Yaskawa INFORM job: OK_R2_O27-28(-60,-90)OKKR.JBI

/JOB
//NAME OK_R2_O27-28(-60,-90)OKKR
///FOLDERNAME X4
//POS
///NPOS 257,257,257,8,0,0
///TOOL 0
///POSTYPE PULSE
///PULSE
C00000=-3986,-112829,-111510,7465,89684,-2966
C00001=-141364,-59194,-77930,23847,91990,-48786
C00002=-141063,-58232,-69990,23735,87869,-49501
C00003=-140498,-58627,-69073,23636,87005,-49471
C00004=-140498,-58696,-68045,23642,86390,-49593
C00005=-140498,-58689,-68203,23640,86482,-49574
C00006=-139283,-59279,-68522,23418,86041,-49222
C00007=-140498,-58679,-68345,23640,86568,-49558
C00008=-140498,-58443,-70820,23629,88081,-49258
C00009=-127873,-62764,-73114,21064,83986,-45532
C00010=-126392,-63087,-72194,20752,82931,-45191
C00011=-125308,-63227,-72265,20505,82639,-44857
C00012=-125876,-63157,-72230,20635,82791,-45032
C00013=-125876,-63224,-70878,20668,81976,-45171
C00014=-126013,-60778,-71127,20647,83335,-44988
C00015=-126013,-60882,-69659,20681,82436,-45141
C00016=-127370,-60434,-72326,20932,84528,-45261
C00017=-126178,-37548,-64770,20629,90906,-43754
C00018=-125360,-36121,-63262,20430,90533,-43541
C00019=-124562,-36215,-63320,20235,90337,-43305
C00020=-125156,-36149,-63276,20379,90482,-43482
C00021=-125105,-34567,-61617,20363,90274,-43498
C00022=-125156,-36149,-63276,20379,90482,-43482
C00023=-135815,-54991,-80141,22838,93753,-46517
C00024=-126128,-100939,-98074,-7833,62391,34723
C00025=-121019,-58487,-70527,-23750,81541,54822
C00026=-122085,-55123,-66318,-23503,80455,54653
C00027=-122085,-55198,-65243,-23545,79813,54780
C00028=-122085,-55189,-65403,-23539,79908,54761
C00029=-123392,-55124,-65366,-23193,79559,54356
C00030=-122085,-54853,-68645,-23426,81902,54365
C00031=-134552,-52582,-66238,-19865,78414,50556
C00032=-135818,-52234,-64976,-19512,77552,50249
C00033=-136587,-51927,-64802,-19268,77420,49997
C00034=-135954,-52181,-64946,-19469,77528,50205
C00035=-135954,-52277,-63949,-19514,76901,50308
C00036=-136080,-52138,-64861,-19432,77470,50170
C00037=-136080,-52251,-63636,-19487,76702,50295
C00038=-135954,-52187,-64889,-19472,77492,50211
C00039=-133506,-28182,-57356,-19912,85326,49780
C00040=-133698,-26913,-56229,-19853,85243,49729
C00041=-134401,-26653,-56048,-19633,85105,49516
C00042=-133766,-26888,-56212,-19832,85229,49708
C00043=-133683,-26061,-55050,-19864,84975,49778
C00044=-133766,-26888,-56212,-19832,85229,49708
C00045=-118022,-32997,-63083,-24386,90185,54129
C00046=-121676,-92941,-80647,-24717,48269,48100
C00047=-126104,-89968,-74727,-22625,45053,46752
C00048=-126437,-97824,-79818,-22747,44125,46828
C00049=-122563,-90224,-74830,-24996,46013,48290
C00050=-126668,-97900,-73203,-24411,40283,47817
C00051=-125704,-63387,-70361,-17497,77836,40931
C00052=-124997,-29881,-53878,-19439,104666,37001
C00053=-125884,-60589,-72245,-19026,100228,37410
C00054=-128512,-118388,-89616,-19043,55419,43468
C00055=-135431,-142346,-71459,-72171,9437,70233
C00056=-131754,-155096,-83372,-71140,11907,70394
C00057=-142652,-70242,-76718,-4199,55092,38367
C00058=-144604,-67983,-72835,-2974,53782,37623
C00059=-145152,-70837,-74169,-2632,53116,37415
C00060=-145458,-72223,-74577,-2444,52646,37302
C00061=-149846,-88596,-70971,7115,30316,34609
C00062=-154437,-99635,-68231,16252,23743,29866
C00063=-154437,-99624,-68210,16257,23736,29864
C00064=-147075,-80257,-74853,-4272,57747,36179
C00065=-135105,-30448,-54067,-19922,99128,39315
C00066=-136639,-45484,-63511,-20526,99341,42271
C00067=-135372,-63496,-79310,-18587,95300,36150
C00068=-132445,-62328,-82142,-19075,98166,36710
C00069=-146017,-78257,-86482,14597,77172,-40405
C00070=-148450,-84312,-78135,27735,61043,-43185
C00071=-146415,-83246,-79022,27034,61486,-42173
C00072=-149676,-80485,-74368,28759,61288,-43622
C00073=-146415,-82526,-75268,27520,59752,-42632
C00074=-148666,-91519,-74847,29905,56218,-44658
C00075=-148661,-91510,-74815,29908,56203,-44660
C00076=-141622,-55635,-68822,15914,88047,-36263
C00077=-139223,-29516,-55234,13545,105159,-43741
C00078=-138881,-22432,-50139,13428,110509,-48714
C00079=-142652,-51115,-68560,12963,107777,-50366
C00080=-150767,-106394,-89377,20632,70658,-55438
C00081=-159311,-126903,-88538,34684,53320,-63895
C00082=-162771,-130732,-86957,36938,52328,-66028
C00083=-169268,-142526,-99377,37807,56354,-67589
C00084=-135427,-86810,-88528,19455,64054,-50570
C00085=-130773,-34503,-67642,16020,92669,-44609
C00086=-128794,-31809,-63686,15472,92294,-44000
C00087=-128893,-32813,-64547,15497,92321,-44030
C00088=-130866,-69048,-76557,19964,64993,-48316
C00089=-131163,-70480,-77226,20153,64757,-48473
C00090=-131351,-74311,-77618,20524,63181,-48835
C00091=-132679,-88532,-78088,22594,56973,-50647
C00092=-132679,-88527,-78070,22596,56965,-50649
C00093=-130794,-63914,-72852,16389,80850,-46075
C00094=-128797,-28836,-55060,14325,107943,-42385
C00095=-129807,-49025,-67626,14097,105546,-43031
C00096=-134716,-44704,-73522,14618,112039,-43955
C00097=-29759,-44704,-73522,14618,112039,-43955
C00098=-57909,-76089,-130518,-12878,65640,73000
C00099=-127209,-68927,-129586,-14791,77681,41071
C00100=-94927,-66213,-124589,-13119,107191,-29169
C00101=-113727,-82793,-127993,9786,99340,-30667
C00102=-113727,-86481,-127524,9719,97186,-30836
C00103=-113727,-85675,-127642,9732,97666,-30798
C00104=-112224,-85220,-127466,9230,97646,-30371
C00105=-92228,-67360,-123883,-12571,107517,-29060
C00106=-93915,-95192,-134825,-11586,99912,-28771
C00107=-93907,-97921,-132985,-11491,97428,-28535
C00108=-94423,-93096,-131262,-11383,98761,-28810
C00109=-93907,-97921,-132985,-11491,97428,-28535
C00110=-98178,-92441,-135596,-10352,101296,-30120
C00111=-110030,-49454,-111281,11211,101949,-41769
C00112=-110030,-52113,-110961,11140,100416,-41912
C00113=-110030,-50840,-111124,11173,101156,-41843
C00114=-108714,-50397,-110891,10661,101109,-41508
C00115=-110030,-50840,-111124,11173,101156,-41843
C00116=-94659,-80928,-124596,-7278,89440,-41621
C00117=-94884,-83616,-122998,-7181,87076,-41547
C00118=-95311,-80232,-121621,-6996,87929,-41716
C00119=-94926,-83537,-124629,-7161,88110,-41617
C00120=-94884,-64304,-125016,-7294,98157,-42187
C00121=-68339,-68740,-122629,-37645,97901,-27341
C00122=-68339,-68740,-122629,-37645,97901,-27341
C00123=-67428,-88828,-131318,-26507,103272,13068
C00124=-71370,-89365,-129778,-25198,101161,12301
C00125=-78547,-84496,-129463,-18628,102671,11282
C00126=-78547,-86342,-129276,-18525,101662,11444
C00127=-78560,-85520,-129334,-18575,102093,11369
C00128=-79372,-81461,-127756,-18419,103003,10989
C00129=-78560,-82342,-129603,-18733,103801,11099
C00130=-72065,-90999,-130386,-24944,100563,12212
C00131=-83791,-78457,-128497,-14695,105981,10194
C00132=-83791,-80329,-128373,-14610,104970,10319
C00133=-83791,-79121,-128456,-14665,105627,10237
C00134=-84464,-75325,-126915,-14548,106502,9937
C00135=-83407,-79441,-129435,-14816,106104,10287
C00136=-72065,-90999,-130386,-24944,100563,12212
C00137=-83702,-92322,-133428,-14376,100027,10952
C00138=-83702,-94820,-133208,-14304,98651,11113
C00139=-83702,-93492,-133334,-14341,99387,11027
C00140=-84690,-87135,-131003,-14116,101025,10548
C00141=-83702,-92262,-133433,-14377,100059,10948
C00142=-70978,-78992,-130158,-26016,106298,11265
C00143=-70978,-75133,-130239,-32870,108132,50816
C00144=-78131,-73748,-122265,-29687,102174,50283
C00145=-78131,-74118,-122214,-29659,101980,50334
C00146=-78131,-76651,-121813,-29472,100626,50691
C00147=-78131,-74997,-122085,-29593,101516,50457
C00148=-79801,-77736,-123237,-28954,100436,50209
C00149=-73940,-85384,-126808,-30662,100615,52053
C00150=-80113,-114247,-134388,-23740,88254,34284
C00151=-81075,-108298,-132442,-23441,89717,33674
C00152=-80541,-110046,-134005,-23615,89911,33813
C00153=-80541,-103654,-135317,-23722,93674,33065
C00154=-68201,-105154,-135623,-27548,96450,36475
C00155=-62711,-72176,-121164,-35654,111043,40715
C00156=-62711,-74449,-120804,-35309,109900,41112
C00157=-62711,-73505,-120963,-35451,110380,40946
C00158=-63747,-76072,-122060,-35030,109506,40878
C00159=-62711,-70908,-121334,-35852,111664,40494
C00160=-49527,-79873,-125116,-38340,114336,44330
C00161=-57136,-119945,-136347,-29907,93340,40844
C00162=-58022,-116776,-135357,-29743,93940,40370
C00163=-57136,-119945,-136347,-29907,93340,40844
C00164=-54754,-67051,-118805,-40417,118327,44687
C00165=-59603,-68009,-118098,-39014,115880,43853
C00166=-69985,-90348,-127433,-28935,99872,36944
C00167=-57627,-107220,-134942,-31595,99953,40891
C00168=-57921,-110194,-135915,-31186,98692,-1554
C00169=-57134,-101414,-130612,-30299,94100,-6411
C00170=-59324,-101870,-130514,-29608,93156,-6916
C00171=-56722,-67413,-112454,-48445,106979,-15822
C00172=-54266,-64565,-109317,-53003,108151,-17088
C00173=-41269,-82198,-112353,-60396,104555,-10877
C00174=-28361,-73162,-108384,-64272,112863,-9833
C00175=-27672,-73415,-108865,-64508,113328,-9806
C00176=-47228,-89020,-130256,-33764,105577,26890
C00177=-61305,-120775,-136286,-22017,83813,21194
C00178=-54809,-66121,-115305,-41444,115205,18852
C00179=-55914,-62658,-119826,-31689,114363,21910
C00180=-59579,-116943,-133527,-40693,98814,56774
C00181=-59579,-111986,-135330,-41226,101614,55657
C00182=-82689,-64404,-114714,-44753,105294,68555
C00183=-85026,-71008,-115277,-43369,102134,69076
C00184=-83828,-73704,-112663,-46568,100432,69183
C00185=-87462,-56287,-104252,-46039,101525,67169
C00186=-100057,-54460,-109437,-30018,101424,67387
C00187=-93453,-70731,-120715,-32763,95417,70730
C00188=-139156,-94805,-132093,18130,87071,69051
C00189=-163867,-98555,-128253,42750,94335,67382
C00190=-172516,-111345,-128204,48282,94494,64723
C00191=-166019,-100240,-124138,46341,91045,66003
C00192=-149033,-114276,-126268,45882,80820,69967
C00193=-120740,-77059,-127423,-1910,96848,70703
C00194=-140122,-66996,-121644,18205,101200,82864
C00195=-124061,-66913,-122683,-715,101740,69762
C00196=-124249,-65814,-122190,-648,101999,69713
C00197=-125559,-65630,-122107,-162,102038,69374
C00198=-119797,-81339,-130415,-2306,92186,71023
C00199=-119797,-76858,-130549,-2315,94569,70980
C00200=-125018,-89354,-136048,304,100400,-3157
C00201=-134660,-90837,-134002,3576,98568,-5831
C00202=-164603,-64987,-122332,34331,112788,-33477
C00203=-154444,-110219,-128747,32478,84481,-37079
C00204=-154411,-110304,-128758,32461,84452,-37077
C00205=-154411,-110304,-128758,32461,84452,-37077
C00206=-154700,-108694,-131145,32499,86507,-36592
C00207=-162794,-57759,-118946,34225,113618,-32605
C00208=-119251,-87160,-133667,-7347,101945,13426
C00209=-129532,-85547,-132715,-6422,100747,15641
C00210=-115912,-82289,-119455,-18954,85425,20858
C00211=-146741,-70967,-114660,-4742,84427,12038
C00212=-151942,-65943,-112379,-2250,85418,10567
C00213=-128583,-88079,-136549,-6779,102009,2369
C00214=-120975,-81846,-133513,-6898,103450,2526
C00215=-155975,-62773,-126766,2743,93886,72191
C00216=-136966,-95819,-134490,20427,86906,86074
C00217=-159533,-96895,-119861,47748,87610,84100
C00218=-155188,-77420,-111739,46252,89058,86685
C00219=-139977,-52066,-108983,28236,100023,90294
C00220=-131749,-86953,-130965,11868,89207,86763
C00221=-130735,-66163,-122382,11485,94387,87521
C00222=-104176,-129682,-135113,-35976,69466,88101
C00223=-103067,-123499,-130669,-38385,71500,88761
C00224=-105160,-95224,-120945,-36174,77532,85788
C00225=-111034,-91676,-120435,-29152,76328,85261
C00226=-109150,-91490,-124842,-29792,79369,85119
C00227=-148549,-77768,-129127,12621,97057,82226
C00228=-138384,-85916,-129968,1380,91848,82299
C00229=-147245,-76344,-125369,14223,97283,83325
C00230=-146767,-75617,-125069,14046,97401,83471
C00231=-145345,-76981,-125634,13486,96870,83803
C00232=-148344,-94092,-136119,12429,93040,81874
C00233=-148344,-94092,-136119,12429,93040,81874
C00234=-149390,-100171,-97789,13457,91429,80931
C00235=-185001,-50343,-102337,59343,112578,87672
C00236=-177996,-87878,-117653,49484,97863,85861
C00237=-172841,-73528,-111525,48418,97852,88154
C00238=-167396,-109795,-125913,40086,79831,90462
C00239=-176701,-106662,-127766,43143,86000,89084
C00240=-178983,-99807,-127488,43897,89483,89622
C00241=-186288,-123588,-135328,46116,87556,34686
C00242=-184402,-113027,-130160,47597,91772,34238
C00243=-190165,-135187,-128789,55315,81887,27042
C00244=-182769,-112039,-115412,62848,86405,24634
C00245=-182898,-80381,-103143,66753,99729,26043
C00246=-184749,-80984,-105447,67423,101319,26279
C00247=-200163,-112982,-117383,65776,95886,23085
C00248=-197571,-143174,-124579,63928,80844,20852
C00249=-197223,-132350,-121232,64115,85612,21537
C00250=-190318,-92922,-107812,68191,103944,23641
C00251=-191351,-89325,-109427,69212,105699,24779
C00252=-198286,-115859,-125385,62599,94515,23403
C00253=-198286,-115859,-125385,62599,94515,23403
C00254=-180994,-114323,-119953,62599,94515,23403
C00255=-7894,-115859,-125385,-1274,91471,-84059
C00256=-4396,-113146,-112965,6547,89872,-11479
BC00000=154740,697504,1071137
BC00001=345717,749885,1074784
BC00002=345717,749885,1074784
BC00003=345717,749885,1074784
BC00004=345717,749885,1074784
BC00005=345717,749885,1074784
BC00006=345717,749885,1074784
BC00007=345717,749885,1074784
BC00008=345717,749885,1074784
BC00009=345717,749885,1074784
BC00010=345717,749885,1074784
BC00011=345717,749885,1074784
BC00012=345717,749885,1074784
BC00013=345717,749885,1074784
BC00014=345717,749885,1074784
BC00015=345717,749885,1074784
BC00016=345717,749885,1074784
BC00017=345717,749885,1074784
BC00018=345717,749885,1074784
BC00019=345717,749885,1074784
BC00020=345717,749885,1074784
BC00021=345717,749885,1074784
BC00022=345717,749885,1074784
BC00023=345717,749885,1074784
BC00024=136436,744253,1074400
BC00025=136436,744253,1074400
BC00026=136435,744254,1074397
BC00027=136435,744254,1074397
BC00028=136435,744254,1074397
BC00029=136435,744254,1074397
BC00030=136435,744254,1074397
BC00031=136435,744254,1074397
BC00032=136435,744254,1074397
BC00033=136435,744254,1074397
BC00034=136435,744254,1074397
BC00035=136435,744254,1074397
BC00036=136435,744254,1074397
BC00037=136435,744254,1074397
BC00038=136435,744254,1074397
BC00039=136435,744254,1074397
BC00040=136435,744254,1074397
BC00041=136435,744254,1074397
BC00042=136435,744254,1074397
BC00043=136435,744254,1074397
BC00044=136435,744254,1074397
BC00045=136435,744254,1074397
BC00046=132140,755225,1075166
BC00047=132140,755225,1075166
BC00048=132140,755225,1075166
BC00049=132140,755225,1075166
BC00050=132141,755225,1075160
BC00051=132140,755225,1075163
BC00052=132140,755225,1075163
BC00053=132140,755225,1075163
BC00054=132140,755225,1075163
BC00055=132140,755225,1075163
BC00056=132140,755225,1075159
BC00057=132140,755225,1075159
BC00058=132140,755225,1075159
BC00059=132140,755225,1075159
BC00060=132140,755225,1075159
BC00061=132140,755225,1075159
BC00062=132140,755225,1075156
BC00063=132140,755225,1075156
BC00064=132140,755225,1075159
BC00065=132140,755225,1075156
BC00066=132140,755225,1075156
BC00067=132140,755225,1075156
BC00068=132140,755225,1075156
BC00069=365187,755225,1075156
BC00070=365187,755225,1075156
BC00071=365187,755225,1075156
BC00072=365187,755225,1075156
BC00073=365187,755225,1075156
BC00074=365187,755225,1075156
BC00075=365187,755225,1075156
BC00076=365187,755225,1075156
BC00077=365187,755225,1075156
BC00078=365187,755225,1075156
BC00079=365187,755225,1075156
BC00080=365187,755225,1075156
BC00081=365187,755225,1075156
BC00082=365187,755225,1075156
BC00083=365187,755225,1075156
BC00084=365187,755225,1075156
BC00085=365187,755225,1075156
BC00086=365187,755225,1075156
BC00087=365187,755225,1075156
BC00088=365187,755225,1075156
BC00089=365187,755225,1075156
BC00090=365187,755225,1075156
BC00091=365187,755225,1075156
BC00092=365187,755225,1075156
BC00093=365187,755225,1075156
BC00094=365187,755225,1075156
BC00095=365187,755225,1075156
BC00096=365187,755225,1075156
BC00097=261045,693732,1070991
BC00098=158970,724604,1070878
BC00099=76284,798681,1075160
BC00100=6539,834987,1075160
BC00101=1106,837815,1075160
BC00102=1106,837815,1075160
BC00103=1106,837815,1075160
BC00104=1106,837815,1075160
BC00105=1106,837815,1075160
BC00106=1106,837815,1075160
BC00107=1106,837815,1075160
BC00108=1106,837815,1075160
BC00109=1106,837815,1075160
BC00110=1106,837815,1075160
BC00111=1106,837815,1075160
BC00112=1106,837815,1075160
BC00113=1106,837815,1075160
BC00114=1106,837815,1075160
BC00115=1106,837815,1075160
BC00116=1106,837815,1075160
BC00117=1106,837815,1075160
BC00118=1106,837815,1075160
BC00119=1106,837815,1075160
BC00120=1106,837815,1075160
BC00121=1106,837815,1075160
BC00122=1106,837815,1075160
BC00123=119538,853346,1061293
BC00124=119538,853346,1061293
BC00125=119538,853346,1061293
BC00126=119539,853345,1061292
BC00127=119538,853346,1061293
BC00128=119538,853346,1061293
BC00129=119538,853346,1061293
BC00130=177839,853346,1064625
BC00131=177839,853346,1061293
BC00132=177839,853346,1061293
BC00133=177839,853346,1061293
BC00134=177839,853346,1061293
BC00135=177839,853346,1061293
BC00136=233775,853346,1064625
BC00137=233775,853794,1058500
BC00138=233775,853794,1058500
BC00139=233775,853794,1058500
BC00140=233774,853794,1058499
BC00141=233775,853794,1058500
BC00142=233775,853794,1059039
BC00143=363355,853794,1059039
BC00144=363355,853794,1059039
BC00145=363355,853794,1059039
BC00146=363355,853794,1059039
BC00147=363355,853794,1059039
BC00148=363355,853794,1059039
BC00149=363355,853794,1059039
BC00150=363355,853794,1059039
BC00151=363355,853794,1059039
BC00152=363355,853794,1059039
BC00153=363355,853794,1059039
BC00154=362752,851033,1059039
BC00155=362481,849794,1059039
BC00156=362481,849794,1059039
BC00157=362481,849794,1059039
BC00158=362481,849794,1059039
BC00159=362481,849794,1059039
BC00160=362481,849794,1059039
BC00161=362481,849794,1059039
BC00162=362481,849794,1059039
BC00163=362481,849794,1059039
BC00164=362481,849794,1059039
BC00165=362481,849794,1059039
BC00166=362481,849794,1059039
BC00167=362481,849794,1059039
BC00168=362482,849793,1059038
BC00169=349829,842790,1059038
BC00170=349829,842790,1059038
BC00171=349829,842790,1059038
BC00172=349829,842790,1059038
BC00173=349829,842790,1059038
BC00174=349829,842790,1059038
BC00175=349829,842790,1059038
BC00176=349829,842790,1059038
BC00177=348819,842790,1059038
BC00178=349829,842790,1059038
BC00179=349829,842790,1059038
BC00180=381424,850930,1066148
BC00181=381424,850930,1066148
BC00182=396386,850930,1066148
BC00183=396386,850930,1066148
BC00184=396386,850930,1066148
BC00185=396386,850930,1066148
BC00186=396386,850930,1066148
BC00187=396386,850930,1066148
BC00188=396386,859792,1066148
BC00189=396386,866222,1066148
BC00190=396386,866222,1066148
BC00191=396386,866222,1066148
BC00192=366433,866054,1066148
BC00193=396386,861777,1066148
BC00194=396386,861777,1066145
BC00195=396386,861777,1066148
BC00196=396386,861777,1066148
BC00197=396386,861777,1066148
BC00198=396386,861777,1066148
BC00199=396386,861777,1066148
BC00200=237377,847193,1066148
BC00201=237377,847194,1066145
BC00202=237377,847194,1066141
BC00203=215951,844802,1066138
BC00204=253673,844832,1066138
BC00205=265455,844832,1066138
BC00206=265455,844832,1066138
BC00207=237377,847194,1066141
BC00208=245654,847194,1066145
BC00209=248473,847194,1066145
BC00210=248473,825286,1066145
BC00211=248473,825343,1066145
BC00212=248473,825343,1066145
BC00213=248473,847194,1066145
BC00214=250700,847194,1066145
BC00215=120403,847194,1066145
BC00216=43580,847194,1066145
BC00217=43580,847194,1066145
BC00218=43580,847194,1066145
BC00219=43580,847194,1066145
BC00220=43579,847194,1066142
BC00221=43579,838034,1066142
BC00222=77368,847082,1066142
BC00223=77368,847082,1066142
BC00224=77368,847082,1066142
BC00225=77368,847082,1066142
BC00226=77368,847082,1066142
BC00227=77368,864301,1066142
BC00228=77367,864301,1066139
BC00229=77368,864301,1066142
BC00230=77368,864301,1066142
BC00231=77368,864301,1066142
BC00232=77368,864301,1066142
BC00233=23315,864301,1066142
BC00234=23830,746014,1066142
BC00235=58368,836918,1066142
BC00236=58368,836918,1066142
BC00237=58368,836918,1066142
BC00238=58368,836918,1066142
BC00239=58368,836918,1066142
BC00240=58368,836918,1066142
BC00241=58368,836918,1066142
BC00242=58368,836918,1066142
BC00243=58368,836918,1066142
BC00244=58368,836918,1066142
BC00245=58368,836918,1066142
BC00246=58368,836918,1066142
BC00247=58368,836918,1066142
BC00248=58368,836918,1066142
BC00249=58368,836918,1066142
BC00250=58368,836918,1066142
BC00251=58368,836918,1066142
BC00252=58368,836918,1066142
BC00253=12933,742434,1066142
BC00254=12933,742434,1066142
BC00255=12933,673240,1066142
BC00256=138860,694957,1070611
EC00000=-454111,-556475
EC00001=-443859,-556475
EC00002=-443859,-556475
EC00003=-443859,-556475
EC00004=-443859,-556475
EC00005=-443859,-556475
EC00006=-443859,-556475
EC00007=-443859,-556475
EC00008=-443859,-556475
EC00009=-443859,-556475
EC00010=-443859,-556475
EC00011=-443859,-556475
EC00012=-443859,-556475
EC00013=-443859,-556475
EC00014=-443859,-556475
EC00015=-443859,-556475
EC00016=-443859,-556475
EC00017=-443859,-556475
EC00018=-443859,-556475
EC00019=-443859,-556475
EC00020=-443859,-556475
EC00021=-443859,-556475
EC00022=-443859,-556475
EC00023=-443859,-556475
EC00024=-444967,-556475
EC00025=-444967,-556475
EC00026=-444965,-556475
EC00027=-444965,-556475
EC00028=-444965,-556475
EC00029=-444965,-556475
EC00030=-444965,-556475
EC00031=-444965,-556475
EC00032=-444965,-556475
EC00033=-444965,-556475
EC00034=-444965,-556475
EC00035=-444965,-556475
EC00036=-444965,-556475
EC00037=-444965,-556475
EC00038=-444965,-556475
EC00039=-444965,-556475
EC00040=-444965,-556475
EC00041=-444965,-556475
EC00042=-444965,-556475
EC00043=-444965,-556475
EC00044=-444965,-556475
EC00045=-444965,-556475
EC00046=-442821,-556475
EC00047=-442821,-556475
EC00048=-442821,-556475
EC00049=-442821,-556475
EC00050=-442817,-556475
EC00051=-442818,-556475
EC00052=-442818,-556475
EC00053=-442818,-556475
EC00054=-442818,-556475
EC00055=-442818,-556475
EC00056=-442816,-556475
EC00057=-442816,-556475
EC00058=-442816,-556475
EC00059=-442816,-556475
EC00060=-442816,-556475
EC00061=-442816,-556475
EC00062=-442815,-556475
EC00063=-442815,-556475
EC00064=-442816,-556475
EC00065=-442814,-556475
EC00066=-442814,-556475
EC00067=-442814,-556475
EC00068=-442814,-556475
EC00069=-442814,-556475
EC00070=-442814,-556475
EC00071=-442814,-556475
EC00072=-442814,-556475
EC00073=-442814,-556475
EC00074=-442814,-556475
EC00075=-442814,-556475
EC00076=-442814,-556475
EC00077=-442814,-556475
EC00078=-442814,-556475
EC00079=-442814,-556475
EC00080=-442814,-556475
EC00081=-442814,-556475
EC00082=-442814,-556475
EC00083=-442814,-556475
EC00084=-442814,-556475
EC00085=-442814,-556475
EC00086=-442814,-556475
EC00087=-442814,-556475
EC00088=-442814,-556475
EC00089=-442814,-556475
EC00090=-442814,-556475
EC00091=-442814,-556475
EC00092=-442814,-556475
EC00093=-442814,-556475
EC00094=-442814,-556475
EC00095=-442814,-556475
EC00096=-442814,-556475
EC00097=-442814,-556475
EC00098=-798155,-556476
EC00099=-798157,-556476
EC00100=-798157,-556476
EC00101=-798157,-556476
EC00102=-798157,-556476
EC00103=-798157,-556476
EC00104=-798157,-556476
EC00105=-798157,-556476
EC00106=-798157,-556476
EC00107=-798157,-556476
EC00108=-798157,-556476
EC00109=-798157,-556476
EC00110=-798157,-556476
EC00111=-798157,-556476
EC00112=-798157,-556476
EC00113=-798157,-556476
EC00114=-798157,-556476
EC00115=-798157,-556476
EC00116=-798157,-556476
EC00117=-798157,-556476
EC00118=-798157,-556476
EC00119=-798157,-556476
EC00120=-798157,-556476
EC00121=-798157,-556476
EC00122=-798157,-556476
EC00123=-798157,-556476
EC00124=-798157,-556476
EC00125=-798157,-556476
EC00126=-798156,-556476
EC00127=-798157,-556476
EC00128=-798157,-556476
EC00129=-798157,-556476
EC00130=-798157,-556476
EC00131=-798157,-556476
EC00132=-798157,-556476
EC00133=-798157,-556476
EC00134=-798157,-556476
EC00135=-798157,-556476
EC00136=-798157,-556476
EC00137=-798157,-556476
EC00138=-798157,-556476
EC00139=-798157,-556476
EC00140=-798155,-556476
EC00141=-798157,-556476
EC00142=-798157,-556476
EC00143=-798157,-556476
EC00144=-798157,-556476
EC00145=-798157,-556476
EC00146=-798157,-556476
EC00147=-798157,-556476
EC00148=-798157,-556476
EC00149=-798157,-556476
EC00150=-798157,-556476
EC00151=-798157,-556476
EC00152=-798157,-556476
EC00153=-798157,-556476
EC00154=-798157,-556476
EC00155=-798157,-556476
EC00156=-798157,-556476
EC00157=-798157,-556476
EC00158=-798157,-556476
EC00159=-798157,-556476
EC00160=-798157,-556476
EC00161=-798157,-556476
EC00162=-798157,-556476
EC00163=-798157,-556476
EC00164=-798157,-556476
EC00165=-798157,-556476
EC00166=-798157,-556476
EC00167=-798157,-556476
EC00168=-798156,-556476
EC00169=-798156,-556476
EC00170=-798156,-556476
EC00171=-798156,-556476
EC00172=-798156,-556476
EC00173=-798156,-556476
EC00174=-798156,-556476
EC00175=-798156,-556476
EC00176=-798156,-556476
EC00177=-798156,-556476
EC00178=-798156,-556476
EC00179=-798156,-556476
EC00180=-798156,-556476
EC00181=-798156,-556476
EC00182=-798156,-556476
EC00183=-798156,-556476
EC00184=-798156,-556476
EC00185=-798156,-556476
EC00186=-798156,-556476
EC00187=-798156,-556476
EC00188=-798156,-556476
EC00189=-798156,-556476
EC00190=-798156,-556476
EC00191=-798156,-556476
EC00192=-798156,-556476
EC00193=-798156,-556476
EC00194=-798155,-556477
EC00195=-798156,-556476
EC00196=-798156,-556476
EC00197=-798156,-556476
EC00198=-798156,-556476
EC00199=-798156,-556476
EC00200=-798156,-556476
EC00201=-798155,-556476
EC00202=-798152,-556477
EC00203=-798150,-556478
EC00204=-798150,-556478
EC00205=-798150,-556478
EC00206=-798150,-556478
EC00207=-798152,-556477
EC00208=-798155,-556476
EC00209=-798155,-556476
EC00210=-798155,-556476
EC00211=-798155,-556476
EC00212=-798155,-556476
EC00213=-798155,-556476
EC00214=-798155,-556476
EC00215=-798155,-556476
EC00216=-798155,-556476
EC00217=-798155,-556476
EC00218=-798155,-556476
EC00219=-798155,-556476
EC00220=-798154,-556476
EC00221=-798154,-556476
EC00222=-798154,-556476
EC00223=-798154,-556476
EC00224=-798154,-556476
EC00225=-798154,-556476
EC00226=-798154,-556476
EC00227=-798154,-556476
EC00228=-798152,-556476
EC00229=-798154,-556476
EC00230=-798154,-556476
EC00231=-798154,-556476
EC00232=-798154,-556476
EC00233=-798154,-556476
EC00234=-798154,-556476
EC00235=-798154,-556476
EC00236=-798154,-556476
EC00237=-798154,-556476
EC00238=-798154,-556476
EC00239=-798154,-556476
EC00240=-798154,-556476
EC00241=-798154,-556476
EC00242=-798154,-556476
EC00243=-798154,-556476
EC00244=-798154,-556476
EC00245=-798154,-556476
EC00246=-798154,-556476
EC00247=-798154,-556476
EC00248=-798154,-556476
EC00249=-798154,-556476
EC00250=-798154,-556476
EC00251=-798154,-556476
EC00252=-798154,-556476
EC00253=-798154,-556476
EC00254=-798154,-556476
EC00255=-798154,-556476
EC00256=0,-556475
///POSTYPE BASE
///RECTAN
///RCONF 0,0,0,0,0,0,0,0,0,0,0,0,0,0,0,0,0,0,0,0,0,0,0,0
P00006=0.222,-3.123,-1.508,0.0000,0.0000,0.0000
P00021=-0.225,-6.128,-0.405,0.0000,0.0000,0.0000
P00022=0.222,-3.123,-1.508,0.0000,0.0000,0.0000
P00023=0.143,-0.036,0.682,0.0000,0.0000,0.0000
P00024=0.145,-0.552,1.326,0.0000,0.0000,0.0000
P00025=-2.003,0.006,0.728,0.0000,0.0000,0.0000
P00026=0.562,-0.002,-0.337,0.0000,0.0000,0.0000
P00027=-0.746,0.015,-9.096,0.0000,0.0000,0.0000
//INST
///DATE 2025/05/21 11:20
///ATTR SC,RW
///GROUP1 RB1,BS1
///GROUP2 ST1
NOP
SFTOF3D
'NOWY PROGRAM KM
SFTOF3D
MOVJ C00000 BC00000 VJ=100.00  +MOVJ EC00000 VJ=100.00
'POMIAR
MOVJ C00001 BC00001 VJ=100.00  +MOVJ EC00001 VJ=100.00
MOVJ C00002 BC00002 VJ=100.00  +MOVJ EC00002 VJ=100.00
SMOVL C00003 BC00003 V=100.0  +MOVJ EC00003
SREFP 3 C00004 BC00004  +REFP EC00004
CALL JOB:SEARCH-R1-S13D
SET P024 P006
SFTON3D P024
SMOVL C00005 BC00005 V=100.0  +MOVJ EC00005
SREFP 3 C00006 BC00006  +REFP EC00006
CALL JOB:SEARCH-R1-S13D
SET P024 P006
SFTON3D P024
SFTOF3D
SMOVL C00007 BC00007 V=166.7  +MOVJ EC00007
MOVJ C00008 BC00008 VJ=100.00  +MOVJ EC00008 VJ=100.00
MOVJ C00009 BC00009 VJ=100.00  +MOVJ EC00009 VJ=100.00
SMOVL C00010 BC00010 V=100.0  +MOVJ EC00010
SREFP 3 C00011 BC00011  +REFP EC00011
CALL JOB:SEARCH-R1-S13D
SET P025 P006
SFTON3D P025
SMOVL C00012 BC00012 V=100.0  +MOVJ EC00012
SREFP 3 C00013 BC00013  +REFP EC00013
CALL JOB:SEARCH-R1-S13D
SET P025 P006
SFTON3D P025
SFTOF3D
SMOVL C00014 BC00014 V=166.7  +MOVJ EC00014
SREFP 3 C00015 BC00015  +REFP EC00015
CALL JOB:SEARCH-R1-S13D
SET P026 P006
SFTON3D P026
SMOVL C00016 BC00016 V=250.0  +MOVJ EC00016
SMOVL C00017 BC00017 V=400.0  +MOVJ EC00017
SMOVL C00018 BC00018 V=100.0  +MOVJ EC00018
SREFP 3 C00019 BC00019  +REFP EC00019
CALL JOB:SEARCH-R1-S13D
SET P026 P006
SFTON3D P026
SMOVL C00020 BC00020 V=100.0  +MOVJ EC00020
SREFP 3 C00021 BC00021  +REFP EC00021
CALL JOB:SEARCH-R1-S13D
SET P026 P006
SFTON3D P026
SMOVL C00022 BC00022 V=166.7  +MOVJ EC00022
MOVJ C00023 BC00023 VJ=100.00  +MOVJ EC00023 VJ=100.00
MOVJ C00024 BC00024 VJ=100.00  +MOVJ EC00024 VJ=100.00
MOVJ C00025 BC00025 VJ=100.00  +MOVJ EC00025 VJ=100.00
SMOVL C00026 BC00026 V=100.0  +MOVJ EC00026
SREFP 3 C00027 BC00027  +REFP EC00027
CALL JOB:SEARCH-R1-S13D
SET P021 P006
SFTON3D P021
SMOVL C00028 BC00028 V=100.0  +MOVJ EC00028
SREFP 3 C00029 BC00029  +REFP EC00029
CALL JOB:SEARCH-R1-S13D
SET P021 P006
SFTON3D P021
SMOVL C00030 BC00030 V=166.7  +MOVJ EC00030
SMOVL C00031 BC00031 V=416.7  +MOVJ EC00031
SMOVL C00032 BC00032 V=100.0  +MOVJ EC00032
SREFP 3 C00033 BC00033  +REFP EC00033
CALL JOB:SEARCH-R1-S13D
SET P021 P006
SFTON3D P021
SMOVL C00034 BC00034 V=100.0  +MOVJ EC00034
SREFP 3 C00035 BC00035  +REFP EC00035
CALL JOB:SEARCH-R1-S13D
SET P021 P006
SFTON3D P021
SFTOF3D
SMOVL C00036 BC00036 V=166.7  +MOVJ EC00036
SREFP 3 C00037 BC00037  +REFP EC00037
CALL JOB:SEARCH-R1-S13D
SET P022 P006
SFTON3D P022
SMOVL C00038 BC00038 V=166.7  +MOVJ EC00038
SMOVL C00039 BC00039 V=416.7  +MOVJ EC00039
SMOVL C00040 BC00040 V=166.7  +MOVJ EC00040
SREFP 3 C00041 BC00041  +REFP EC00041
CALL JOB:SEARCH-R1-S13D
SET P022 P006
SFTON3D P022
SMOVL C00042 BC00042 V=166.7  +MOVJ EC00042
SREFP 3 C00043 BC00043  +REFP EC00043
CALL JOB:SEARCH-R1-S13D
SET P022 P006
SFTON3D P022
SMOVL C00044 BC00044 V=166.7  +MOVJ EC00044
SMOVL C00045 BC00045 V=666.7  +MOVJ EC00045
SFTOF3D
MOVJ C00046 BC00046 VJ=100.00  +MOVJ EC00046 VJ=100.00
MACRO1 MJ#(0) ARGF9
SFTON3D P021
SMOVL C00047 BC00047 V=166.7  +MOVJ EC00047
SREFP 1 C00048 BC00048  +REFP EC00048
SREFP 2 C00049 BC00049  +REFP EC00049
ARCON
SWVON WEV#(13)
SMOVL C00050 BC00050 V=10.0  +MOVJ EC00050
SMOVL C00051 BC00051 V=10.0  +MOVJ EC00051
SMOVL C00052 BC00052 V=8.3  +MOVJ EC00052
SMOVL C00053 BC00053 V=8.3  +MOVJ EC00053
SMOVL C00054 BC00054 V=8.3  +MOVJ EC00054
SMOVL C00055 BC00055 V=10.0  +MOVJ EC00055
ARCOF
SWVOF
SFTOF3D
SMOVL C00056 BC00056 V=250.0  +MOVJ EC00056
SMOVL C00057 BC00057 V=1000.0  +MOVJ EC00057
MACRO1 MJ#(0) ARGF17
SFTON3D P022
SMOVL C00058 BC00058 V=166.7  +MOVJ EC00058
ARCON
SMOVL C00059 BC00059 V=10.0  +MOVJ EC00059
SMOVL C00060 BC00060 V=10.0  +MOVJ EC00060
SMOVL C00061 BC00061 V=9.2  +MOVJ EC00061
SMOVL C00062 BC00062 V=9.2  +MOVJ EC00062
SMOVC C00063 BC00063 V=9.2  +MOVJ EC00063
SMOVC C00064 BC00064 V=9.2  +MOVJ EC00064
SFTON3D P022
SMOVC C00065 BC00065 V=9.2  +MOVJ EC00065
SMOVL C00066 BC00066 V=9.2  +MOVJ EC00066
ARCOF
SMOVL C00067 BC00067 V=166.7  +MOVJ EC00067
SFTOF3D
MOVJ C00068 BC00068 VJ=100.00  +MOVJ EC00068 VJ=100.00
MOVJ C00069 BC00069 VJ=100.00  +MOVJ EC00069 VJ=100.00
MACRO1 MJ#(0) ARGF9
MOVJ C00070 BC00070 VJ=100.00  +MOVJ EC00070 VJ=100.00
SWVON WEV#(13)
SREFP 1 C00071 BC00071  +REFP EC00071
SREFP 2 C00072 BC00072  +REFP EC00072
SFTON3D P024
SMOVL C00073 BC00073 V=166.7  +MOVJ EC00073
ARCON
SMOVL C00074 BC00074 V=10.0  +MOVJ EC00074
SMOVC C00075 BC00075 V=10.0  +MOVJ EC00075
SMOVC C00076 BC00076 V=10.0  +MOVJ EC00076
SMOVC C00077 BC00077 V=10.0  +MOVJ EC00077
SMOVL C00078 BC00078 V=10.0  +MOVJ EC00078
SMOVL C00079 BC00079 V=10.0  +MOVJ EC00079
SMOVL C00080 BC00080 V=10.0  +MOVJ EC00080
SMOVL C00081 BC00081 V=10.0  +MOVJ EC00081
SMOVL C00082 BC00082 V=10.0  +MOVJ EC00082
ARCOF
SWVOF
SMOVL C00083 BC00083 V=400.0  +MOVJ EC00083
SMOVL C00084 BC00084 V=1000.0  +MOVJ EC00084
SMOVL C00085 BC00085 V=1000.0  +MOVJ EC00085
MACRO1 MJ#(0) ARGF17
SFTON3D P026
SMOVL C00086 BC00086 V=166.7  +MOVJ EC00086
ARCON
SMOVL C00087 BC00087 V=9.2  +MOVJ EC00087
SMOVL C00088 BC00088 V=9.2  +MOVJ EC00088
SMOVL C00089 BC00089 V=9.2  +MOVJ EC00089
SMOVL C00090 BC00090 V=9.2  +MOVJ EC00090
SMOVL C00091 BC00091 V=9.2  +MOVJ EC00091
SMOVC C00092 BC00092 V=9.2  +MOVJ EC00092
SMOVC C00093 BC00093 V=9.2  +MOVJ EC00093
SFTON3D P025
SMOVC C00094 BC00094 V=9.2  +MOVJ EC00094
SMOVL C00095 BC00095 V=8.3  +MOVJ EC00095
ARCOF
SFTOF3D
SMOVL C00096 BC00096 V=250.0  +MOVJ EC00096
MOVJ C00097 BC00097 VJ=100.00  +MOVJ EC00097 VJ=100.00
'DRUGA POZYCJA
CALL JOB:CLEAN-R1_KM_NEW
MOVJ C00098 BC00098 VJ=100.00  +MOVJ EC00098 VJ=100.00
MOVJ C00099 BC00099 VJ=100.00  +MOVJ EC00099 VJ=20.00
MOVJ C00100 BC00100 VJ=100.00  +MOVJ EC00100 VJ=100.00
'POMIAR
COMM PAUSE
COMM SMOVL C00101 BC00101 V=100.0  +MOVJ EC00101
COMM SREFP 3 C00102 BC00102  +REFP EC00102
COMM CALL JOB:SEARCH-R1-S13D
COMM SET P021 P006
COMM SFTON3D P021
COMM SMOVL C00103 BC00103 V=100.0  +MOVJ EC00103
COMM SREFP 3 C00104 BC00104  +REFP EC00104
COMM CALL JOB:SEARCH-R1-S13D
COMM SET P021 P006
COMM SFTON3D P021
COMM SMOVL C00105 BC00105 V=100.0  +MOVJ EC00105
COMM SMOVL C00106 BC00106 V=100.0  +MOVJ EC00106
COMM SMOVL C00107 BC00107 V=100.0  +MOVJ EC00107
COMM SREFP 3 C00108 BC00108  +REFP EC00108
COMM CALL JOB:SEARCH-R1-S13D
COMM SET P021 P006
COMM SFTON3D P021
COMM SFTOF3D
COMM SMOVL C00109 BC00109 V=100.0  +MOVJ EC00109
COMM SMOVL C00110 BC00110 V=100.0  +MOVJ EC00110
COMM 'POMIAR2
SMOVL C00111 BC00111 V=100.0  +MOVJ EC00111
SREFP 3 C00112 BC00112  +REFP EC00112
CALL JOB:SEARCH-R1-S13D
SET P022 P006
SFTON3D P022
SMOVL C00113 BC00113 V=100.0  +MOVJ EC00113
SREFP 3 C00114 BC00114  +REFP EC00114
CALL JOB:SEARCH-R1-S13D
SET P022 P006
SFTON3D P022
SMOVL C00115 BC00115 V=100.0  +MOVJ EC00115
SMOVL C00116 BC00116 V=100.0  +MOVJ EC00116
SMOVL C00117 BC00117 V=100.0  +MOVJ EC00117
SREFP 3 C00118 BC00118  +REFP EC00118
CALL JOB:SEARCH-R1-S13D
SET P022 P006
SFTON3D P022
SFTOF3D
SMOVL C00119 BC00119 V=100.0  +MOVJ EC00119
SMOVL C00120 BC00120 V=100.0  +MOVJ EC00120
SMOVL C00121 BC00121 V=100.0  +MOVJ EC00121
MOVJ C00122 BC00122 VJ=20.00  +MOVJ EC00122 VJ=20.00
MOVJ C00123 BC00123 VJ=50.00  +MOVJ EC00123 VJ=20.00
SMOVL C00124 BC00124 V=100.0  +MOVJ EC00124
'POMIAR3
SMOVL C00125 BC00125 V=100.0  +MOVJ EC00125
SREFP 3 C00126 BC00126  +REFP EC00126
CALL JOB:SEARCH-R1-S13D
SET P023 P006
SFTON3D P023
SMOVL C00127 BC00127 V=100.0  +MOVJ EC00127
SREFP 3 C00128 BC00128  +REFP EC00128
CALL JOB:SEARCH-R1-S13D
SET P023 P006
SFTON3D P023
SMOVL C00129 BC00129 V=100.0  +MOVJ EC00129
'POMIAR4
MOVJ C00130 BC00130 VJ=50.00  +MOVJ EC00130 VJ=20.00
SMOVL C00131 BC00131 V=100.0  +MOVJ EC00131
SREFP 3 C00132 BC00132  +REFP EC00132
CALL JOB:SEARCH-R1-S13D
SET P024 P006
SFTON3D P024
SMOVL C00133 BC00133 V=100.0  +MOVJ EC00133
SREFP 3 C00134 BC00134  +REFP EC00134
CALL JOB:SEARCH-R1-S13D
SET P024 P006
SFTON3D P024
SMOVL C00135 BC00135 V=100.0  +MOVJ EC00135
SFTOF3D
'POMIAR5
MOVJ C00136 BC00136 VJ=50.00  +MOVJ EC00136 VJ=20.00
SMOVL C00137 BC00137 V=100.0  +MOVJ EC00137
SREFP 3 C00138 BC00138  +REFP EC00138
CALL JOB:SEARCH-R1-S13D
SET P025 P006
SFTON3D P025
SMOVL C00139 BC00139 V=100.0  +MOVJ EC00139
SREFP 3 C00140 BC00140  +REFP EC00140
CALL JOB:SEARCH-R1-S13D
SET P025 P006
SFTON3D P025
SMOVL C00141 BC00141 V=100.0  +MOVJ EC00141
SMOVL C00142 BC00142 V=250.0  +MOVJ EC00142
MOVJ C00143 BC00143 VJ=50.00  +MOVJ EC00143 VJ=20.00
SMOVL C00144 BC00144 V=250.0  +MOVJ EC00144
SFTOF3D
'POMIAR6
SMOVL C00145 BC00145 V=100.0  +MOVJ EC00145
SREFP 3 C00146 BC00146  +REFP EC00146
CALL JOB:SEARCH-R1-S13D
SET P026 P006
SFTON3D P026
SMOVL C00147 BC00147 V=100.0  +MOVJ EC00147
SREFP 3 C00148 BC00148  +REFP EC00148
CALL JOB:SEARCH-R1-S13D
SET P026 P006
SFTON3D P026
SMOVL C00149 BC00149 V=100.0  +MOVJ EC00149
SMOVL C00150 BC00150 V=100.0  +MOVJ EC00150
SREFP 3 C00151 BC00151  +REFP EC00151
CALL JOB:SEARCH-R1-S13D
SET P026 P006
SFTON3D P026
SMOVL C00152 BC00152 V=100.0  +MOVJ EC00152
SMOVL C00153 BC00153 V=166.7  +MOVJ EC00153
SMOVL C00154 BC00154 V=166.7  +MOVJ EC00154
SFTOF3D
COMM PAUSE
COMM 'POMIAR7
COMM SMOVL C00155 BC00155 V=100.0  +MOVJ EC00155
COMM SREFP 3 C00156 BC00156  +REFP EC00156
COMM CALL JOB:SEARCH-R1-S13D
COMM SET P027 P006
COMM SFTON3D P027
COMM SMOVL C00157 BC00157 V=100.0  +MOVJ EC00157
COMM SREFP 3 C00158 BC00158  +REFP EC00158
COMM CALL JOB:SEARCH-R1-S13D
COMM SET P027 P006
COMM SFTON3D P027
COMM SMOVL C00159 BC00159 V=100.0  +MOVJ EC00159
COMM SMOVL C00160 BC00160 V=133.3  +MOVJ EC00160
COMM SMOVL C00161 BC00161 V=100.0  +MOVJ EC00161
COMM SREFP 3 C00162 BC00162  +REFP EC00162
COMM CALL JOB:SEARCH-R1-S13D
COMM SET P027 P006
COMM SFTON3D P027
COMM SMOVL C00163 BC00163 V=100.0  +MOVJ EC00163
COMM SFTOF3D
COMM 'SPAWANIE
COMM MACRO1 MJ#(0) ARGF6
COMM SMOVL C00164 BC00164 V=166.7  +MOVJ EC00164
COMM SFTON3D P027
COMM SMOVL C00165 BC00165 V=133.3  +MOVJ EC00165
COMM ARCON
COMM SMOVL C00166 BC00166 V=8.3  +MOVJ EC00166
COMM ARCOF
COMM SMOVL C00167 BC00167 V=166.7  +MOVJ EC00167
COMM SMOVL C00168 BC00168 V=166.7  +MOVJ EC00168
COMM SMOVL C00169 BC00169 V=166.7  +MOVJ EC00169
COMM ARCON
COMM SMOVL C00170 BC00170 V=8.3  +MOVJ EC00170
COMM SMOVL C00171 BC00171 V=8.3  +MOVJ EC00171
COMM SMOVL C00172 BC00172 V=8.3  +MOVJ EC00172
COMM ARCOF
COMM SMOVL C00173 BC00173 V=166.7  +MOVJ EC00173
COMM SMOVL C00174 BC00174 V=166.7  +MOVJ EC00174
COMM MOVJ C00175 BC00175 VJ=20.00  +MOVJ EC00175 VJ=20.00
COMM MOVJ C00176 BC00176 VJ=40.00  +MOVJ EC00176 VJ=20.00
COMM MACRO1 MJ#(0) ARGF6
COMM SMOVL C00177 BC00177 V=133.3  +MOVJ EC00177
COMM ARCON
COMM SMOVL C00178 BC00178 V=13.3  +MOVJ EC00178
COMM ARCOF
COMM SFTOF3D
COMM SMOVL C00179 BC00179 V=166.7  +MOVJ EC00179
COMM SMOVL C00180 BC00180 V=333.3  +MOVJ EC00180
COMM PAUSE
MOVJ C00181 BC00181 VJ=100.00  +MOVJ EC00181 VJ=20.00
MOVJ C00182 BC00182 VJ=100.00  +MOVJ EC00182 VJ=20.00
SMOVL C00183 BC00183 V=183.3  +MOVJ EC00183
SFTON3D P026
MACRO1 MJ#(0) ARGF21
SMOVL C00184 BC00184 V=133.3  +MOVJ EC00184
ARCON
SMOVL C00185 BC00185 V=10.0  +MOVJ EC00185
SMOVL C00186 BC00186 V=10.0  +MOVJ EC00186
ARCOF
SMOVL C00187 BC00187 V=250.0  +MOVJ EC00187
SMOVL C00188 BC00188 V=250.0  +MOVJ EC00188
SMOVL C00189 BC00189 V=250.0  +MOVJ EC00189
SFTON3D P026
SMOVL C00190 BC00190 V=133.3  +MOVJ EC00190
ARCON
SMOVL C00191 BC00191 V=9.2  +MOVJ EC00191
SMOVL C00192 BC00192 V=10.0  +MOVJ EC00192
ARCOF
SMOVL C00193 BC00193 V=83.3  +MOVJ EC00193
SFTON3D P026
SMOVL C00194 BC00194 V=83.3  +MOVJ EC00194
ARCON
SWVON WEV#(103)
SMOVL C00195 BC00195 V=8.3  +MOVJ EC00195
SMOVL C00196 BC00196 V=9.2  +MOVJ EC00196
SMOVL C00197 BC00197 V=9.2  +MOVJ EC00197
ARCOF
SWVOF
SFTOF3D
SMOVL C00198 BC00198 V=250.0  +MOVJ EC00198
MOVJ C00199 BC00199 VJ=100.00  +MOVJ EC00199 VJ=20.00
MOVJ C00200 BC00200 VJ=80.00  +MOVJ EC00200 VJ=20.00
MOVJ C00201 BC00201 VJ=80.00  +MOVJ EC00201 VJ=20.00
MACRO1 MJ#(0) ARGF14
MOVJ C00202 BC00202 VJ=20.00  +MOVJ EC00202 VJ=0.78
SFTON3D P024
SMOVL C00203 BC00203 V=166.7 PL=0  +MOVJ EC00203
ARCON
SFTON3D P025
SMOVL C00204 BC00204 V=11.7  +MOVJ EC00204
SMOVL C00205 BC00205 V=11.7  +MOVJ EC00205
ARCOF
SMOVL C00206 BC00206 V=166.7  +MOVJ EC00206
SFTOF3D
MOVJ C00207 BC00207 VJ=20.00  +MOVJ EC00207 VJ=20.00
SMOVL C00208 BC00208 V=250.0  +MOVJ EC00208
SMOVL C00209 BC00209 V=166.7  +MOVJ EC00209
SFTON3D P024
SMOVL C00210 BC00210 V=166.7 PL=0  +MOVJ EC00210
ARCON
SFTON3D P023
SMOVL C00211 BC00211 V=11.7  +MOVJ EC00211
SMOVL C00212 BC00212 V=11.7  +MOVJ EC00212
ARCOF
SFTOF3D
SMOVL C00213 BC00213 V=250.0  +MOVJ EC00213
MOVJ C00214 BC00214 VJ=100.00  +MOVJ EC00214 VJ=20.00
MOVJ C00215 BC00215 VJ=100.00  +MOVJ EC00215 VJ=20.00
MOVJ C00216 BC00216 VJ=100.00  +MOVJ EC00216 VJ=20.00
MACRO1 MJ#(0) ARGF21
SFTON3D P022
SMOVL C00217 BC00217 V=250.0  +MOVJ EC00217
ARCON
SMOVL C00218 BC00218 V=9.2  +MOVJ EC00218
SMOVL C00219 BC00219 V=10.0  +MOVJ EC00219
ARCOF
SMOVL C00220 BC00220 V=200.0  +MOVJ EC00220
SMOVL C00221 BC00221 V=166.7  +MOVJ EC00221
SMOVL C00222 BC00222 V=166.7  +MOVJ EC00222
SMOVL C00223 BC00223 V=133.3  +MOVJ EC00223
ARCON
SMOVL C00224 BC00224 V=9.2  +MOVJ EC00224
SMOVL C00225 BC00225 V=10.0  +MOVJ EC00225
ARCOF
SMOVL C00226 BC00226 V=166.7  +MOVJ EC00226
SMOVL C00227 BC00227 V=166.7  +MOVJ EC00227
SMOVL C00228 BC00228 V=133.3  +MOVJ EC00228
ARCON
SWVON WEV#(103)
SMOVL C00229 BC00229 V=8.3  +MOVJ EC00229
SMOVL C00230 BC00230 V=9.2  +MOVJ EC00230
SMOVL C00231 BC00231 V=9.2  +MOVJ EC00231
ARCOF
SWVOF
SMOVL C00232 BC00232 V=166.7  +MOVJ EC00232
SFTOF3D
MOVL C00233 BC00233 V=416.7  +MOVJ EC00233 VJ=0.78
MOVL C00234 BC00234 V=416.7  +MOVJ EC00234 VJ=0.78
COMM PAUSE
COMM SMOVL C00235 BC00235 V=166.7  +MOVJ EC00235
COMM MACRO1 MJ#(0) ARGF6
COMM SFTON3D P021
COMM SMOVL C00236 BC00236 V=133.3  +MOVJ EC00236
COMM ARCON
COMM SMOVL C00237 BC00237 V=8.3  +MOVJ EC00237
COMM SMOVL C00238 BC00238 V=8.3  +MOVJ EC00238
COMM ARCOF
COMM SMOVL C00239 BC00239 V=133.3  +MOVJ EC00239
COMM MOVJ C00240 BC00240 VJ=20.00  +MOVJ EC00240 VJ=20.00
COMM MOVJ C00241 BC00241 VJ=100.00  +MOVJ EC00241 VJ=20.00
COMM MOVJ C00242 BC00242 VJ=100.00  +MOVJ EC00242 VJ=20.00
COMM SMOVL C00243 BC00243 V=66.7  +MOVJ EC00243
COMM ARCON
COMM SMOVL C00244 BC00244 V=8.3  +MOVJ EC00244
COMM SMOVL C00245 BC00245 V=8.3  +MOVJ EC00245
COMM ARCOF
COMM MOVJ C00246 BC00246 VJ=20.00  +MOVJ EC00246 VJ=20.00
COMM MOVJ C00247 BC00247 VJ=100.00  +MOVJ EC00247 VJ=20.00
COMM MACRO1 MJ#(0) ARGF6
COMM SMOVL C00248 BC00248 V=100.0  +MOVJ EC00248
COMM ARCON
COMM SMOVL C00249 BC00249 V=13.3  +MOVJ EC00249
COMM SMOVL C00250 BC00250 V=13.3  +MOVJ EC00250
COMM ARCOF
COMM SFTOF3D
COMM SMOVL C00251 BC00251 V=166.7  +MOVJ EC00251
COMM SMOVL C00252 BC00252 V=250.0  +MOVJ EC00252
SMOVL C00253 BC00253 V=1000.0  +MOVJ EC00253
MOVJ C00254 BC00254 VJ=100.00  +MOVJ EC00254 VJ=100.00
MOVJ C00255 BC00255 VJ=100.00  +MOVJ EC00255 VJ=20.00
MOVJ C00256 BC00256 VJ=100.00  +MOVJ EC00256 VJ=100.00
END
